// TwinCAT 3 PLC project PLC_project
// ProgramVersion: 3.1.4023.0
// libraries:
//   Tc2_Standard, * (Beckhoff Automation GmbH)
//   Tc2_System, * (Beckhoff Automation GmbH)
//   Tc3_Module, * (Beckhoff Automation GmbH)
//   Tc3_Vision, * (Beckhoff Automation GmbH)
// project tree:
//   / PlcTask.TcTTO
//   POUs/ MAIN.TcPOU
// real-time tasks:
//   TASK VnTask ImgAcq (FileSource1): cycle T#10ms, priority 5, ADS port 350
//   TASK PlcTask: cycle T#10ms, priority 20, ADS port 351

CONFIGURATION PLC_project
    RESOURCE PLC ON TwinCAT3
        TASK PlcTask(INTERVAL := T#10ms, PRIORITY := 20);
        PROGRAM MAIN WITH PlcTask : MAIN;
    END_RESOURCE
END_CONFIGURATION

// ---- POUs/MAIN.TcPOU
PROGRAM MAIN
VAR
	hr							:	HRESULT;
	fbCamera					:	FB_VN_FileSourceControl; //For cameras FB_VN_SimpleCameraControl instead
	eState						:	ETcVnCameraState;
	ipImageIn					:	ITcVnImage;
	ipProcessedImage			:	ITcVnImage;
	REFipProcessedImage  		: 	REFERENCE TO ITcVnImage;
	ipImageInDisplay			:	ITcVnDisplayableImage;
	ipProcessedImageToDisplay	:	ITcVnDisplayableImage;
	nNewImageCounter			:   UINT;
	
	// Put text variables
	text: STRING:='TEST';
	x: UDINT:=100;
	y: UDINT:=100;
	scaleFont: LREAL:=1;
	
	
	// Write image variables
	fbWriteImage         :   FB_VN_WriteImage := (nTimeout := T#500MS); 
	sFilePath            :   STRING(255) := '';
	bWriteImageTrigger   :   BOOL;
	bWriteImageWaitResult:   BOOL;
	bWriteImageDone      :   BOOL;
	nReturnCode          :   UDINT;

END_VAR

eState:=fbCamera.GetState();

IF eState = TCVN_CS_ERROR THEN
	hr:=fbCamera.Reset();
	
ELSIF eState<TCVN_CS_ACQUIRING THEN 
	hr:=fbCamera.StartAcquisition();
	
ELSIF eState=TCVN_CS_ACQUIRING THEN 
	hr:=fbCamera.GetCurrentImage(ipImageIn);
	
	IF SUCCEEDED(hr) AND ipImageIn<>0 THEN	
		//Write label
		REFipProcessedImage REF= ipProcessedImage;
		F_VN_CopyImage(ipImageIn,REFipProcessedImage,hr);
	
		hr := F_VN_PutLabel(
    		sText     		:=  text,
    		ipDestImage     :=  ipProcessedImage,
    		nX      		:=  x, 
    		nY       		:=  y, 
   			fFontScale  	:=  scaleFont,
    		hrPrev          :=  hr
		);
		
		IF NOT fbWriteImage.bBusy AND bWriteImageTrigger THEN
        	bWriteImageTrigger := FALSE;
        	bWriteImageDone := FALSE;
       		bWriteImageWaitResult := TRUE;

        	// With setting sFilePath:= '' to an empty string the images are saved under the default path
        	// The default path can be set at the service configuration tab of the Vision Node
        	// If sFilePath is set, it must contain the full path, image name and type
        	// for example: sFilePath := 'C:\WriteImage\ImageName.bmp'
        	fbWriteImage(ipImage := REFipProcessedImage, sFilePath := sFilePath, bWrite := TRUE);
    	END_IF
		
		hr:=F_VN_TransformIntoDisplayableImage(ipImageIn,ipImageInDisplay,hr);
		hr:=F_VN_TransformIntoDisplayableImage(ipProcessedImage,ipProcessedImageToDisplay,hr);
	END_IF
	
END_IF


fbWriteImage(sFilepath:= '', bWrite := FALSE);

IF bWriteImageWaitResult AND NOT fbWriteImage.bBusy THEN
    bWriteImageWaitResult := FALSE;
    // Check if fbWriteImage was finished successfully or implement error handling
    IF fbWriteImage.bError THEN
        nReturnCode := fbWriteImage.nErrorId AND 16#FFF;
    ELSE
        bWriteImageDone := TRUE;
        nReturnCode := 0;
    END_IF
END_IF

END_PROGRAM
